FUNCTION_BLOCK _LINT_TestSuite EXTENDS TcUnit.FB_TestSuite
VAR
END_VAR

TestAddress();
TestClearReference();
TestClone();
TestTypeNameReturnsExpected();
TestIsFloat();
TestIsSigned();
TestMakeReferenceToFollowsReference();
TestMakeReferenceToUpdatesReference();
TestSize();
TestValueReturnsExpectedAfterInit();
TestValueReturnsExpectedAfterChange();
TestSerializeTypeWith();
TestSerializeWith();
TestTryDeserializeFrom();
TestTryMakeReferenceToFollowsReference();
TestTryMakeReferenceToUpdatesReference();

METHOD PUBLIC TestAddress
VAR
    _type : _LINT(0);
    notExpected : PVOID := 0;
    actual : PVOID;
END_VAR
TEST('TestAddress');

actual := _type.Address;

AssertFalse(
    Condition := (notExpected = actual),
    Message := 'Type did not return a valid address.'
);

TEST_FINISHED();
END_METHOD

METHOD PUBLIC TestClearReference
VAR
    _type : _LINT(0);
	target : LINT := 0;
    expected : LINT := 0;
    actual : LINT;
END_VAR
TEST('TestClearReference');

_type.MakeReferenceTo(target);
_type.ClearReference();
target := 123;

actual := _type.Value;

AssertEquals(
    Expected := expected,
    Actual := actual,
    Message := 'Value incorrectly followed target change'
);

TEST_FINISHED();
END_METHOD

METHOD PUBLIC TestClone
VAR
    _type : _LINT(123);
	clone : I_Datatype;
	isValidClone : BOOL;
	compareResult : DINT;
END_VAR
TEST('TestClone');

clone := _type.Clone();

isValidClone := clone <> 0;

IF isValidClone THEN
	compareResult := memcmp(_type.Address, clone.Address, clone.Size);
END_IF

AssertTrue(
	Condition := isValidClone,
	Message := 'Clone did not produce a clone'
);

AssertEquals_DINT(
	Expected := 0,
    Actual := compareResult,
    Message := 'Clone did not return a valid clone.'
);

clone.Dispose();

TEST_FINISHED();
END_METHOD

METHOD PUBLIC TestIsFloat
VAR
    _type : _LINT(0);
END_VAR
TEST('TestIsFloat');

AssertFalse(
	Condition := _type.IsFloat,
    Message := 'Type did not correctly identify itself as being unsigned'
);

TEST_FINISHED();
END_METHOD

METHOD PUBLIC TestIsSigned
VAR
    _type : _LINT(0);
END_VAR
TEST('TestIsSigned');

AssertTrue(
	Condition := _type.IsSigned,
    Message := 'Type did not correctly identify itself as being signed'
);

TEST_FINISHED();
END_METHOD

METHOD PUBLIC TestMakeReferenceToFollowsReference
VAR
    _type : _LINT(0);
	target : LINT := 0;
    expected : LINT := 123;
    actual : LINT;
END_VAR
TEST('TestMakeReferenceToFollowsReference');

_type.MakeReferenceTo(target);
target := 123;

actual := _type.Value;

AssertEquals(
    Expected := expected,
    Actual := actual,
    Message := 'Value did not follow target change'
);

TEST_FINISHED();
END_METHOD

METHOD PUBLIC TestMakeReferenceToUpdatesReference
VAR
    _type : _LINT(0);
	target : LINT := 0;
    expected : LINT := 123;
    actual : LINT;
END_VAR
TEST('TestMakeReferenceToUpdatesReference');

_type.MakeReferenceTo(target);
_type.Value := 123;

actual := target;

AssertEquals(
    Expected := expected,
    Actual := actual,
    Message := 'Value did not update target'
);

TEST_FINISHED();
END_METHOD

METHOD PUBLIC TestSerializeTypeWith
VAR
    _type : _LINT(0);
    serializer : JsonSerializer;
    expected : STRING(500) := '{"typeName":"LINT","minValue":-9223372036854775808,"maxValue":9223372036854775807,"isSigned":true,"isFloat":false}';
    actual : STRING(500);
END_VAR
TEST('TestSerializeTypeWith');

serializer.Reset();
_type.SerializeTypeWith(serializer);
serializer.TryGetSerializedData(ADR(actual), SIZEOF(actual));

AssertEquals_STRING(
    Expected := expected,
    Actual := actual,
    Message := 'Serialization of type did not return correct string.'
);

TEST_FINISHED();
END_METHOD

METHOD PUBLIC TestSerializeWith
VAR
    _type : _LINT(32767);
    serializer : JsonSerializer;
    expected : STRING := '32767';
    actual : STRING(500);
END_VAR
TEST('TestSerializeWith');

serializer.Reset();
_type.SerializeWith(serializer);
serializer.TryGetSerializedData(ADR(actual), SIZEOF(actual));

AssertEquals_STRING(
    Expected := expected,
    Actual := actual,
    Message := 'Serialization of type data did not return correct string.'
);

TEST_FINISHED();
END_METHOD

METHOD PUBLIC TestSize
VAR
    _type : _LINT(0);
    expected : UDINT := SIZEOF(LINT);
    actual : UDINT;
END_VAR
TEST('TestSize');

actual := _type.Size;

AssertEquals_UDINT(
    Expected := Expected,
    Actual := actual,
    Message := 'Type did not return the correct size.'
);

TEST_FINISHED();
END_METHOD

METHOD PUBLIC TestTryDeserializeFrom
VAR
    deserializer : JsonDeserializer;
    feedback : DeserializerFeedback;
    json : STRING := '32767';
    _type : _LINT(0);
    expected : LINT := 32767;
    actual : LINT;
 END_VAR
TEST('TestTryDeserializeFrom');

deserializer.Reset();
deserializer.TryLoad(json);
_type.TryDeserializeFrom(Deserializer, Feedback);

actual := _type.Value;

AssertEquals(
    Expected := expected,
    Actual := actual,
    Message := 'Type did not deserialize correctly.'
);

TEST_FINISHED();
END_METHOD

METHOD PUBLIC TestTryMakeReferenceToFollowsReference
VAR
    _type : _LINT(0);
	target : _LINT(0);
    expected : LINT := 123;
    actual : LINT;
END_VAR
TEST('TestTryMakeReferenceToFollowsReference');

_type.TryMakeReferenceTo(target);
target.Value := 123;

actual := _type.Value;

AssertEquals(
    Expected := expected,
    Actual := actual,
    Message := 'Value did not follow target change'
);

TEST_FINISHED();
END_METHOD

METHOD PUBLIC TestTryMakeReferenceToUpdatesReference
VAR
    _type : _LINT(0);
	target : _LINT(0);
    expected : LINT := 123;
    actual : LINT;
END_VAR
TEST('TestTryMakeReferenceToUpdatesReference');

_type.TryMakeReferenceTo(target);
_type.Value := 123;

actual := target.Value;

AssertEquals(
    Expected := expected,
    Actual := actual,
    Message := 'Value did not update target'
);

TEST_FINISHED();
END_METHOD

METHOD PUBLIC TestTypeNameReturnsExpected
VAR
    _type : _LINT(0);
    expected : STRING := 'LINT';
    actual : STRING;
END_VAR
TEST('TestTypeNameReturnsExpected');

actual := _type.TypeName;

AssertEquals_STRING(
    Expected := expected,
    Actual := actual,
    Message := 'Type did not return correct iec type.'
);

TEST_FINISHED();
END_METHOD

METHOD PUBLIC TestValueReturnsExpectedAfterChange
VAR
    _type : _LINT(0);
    expected : LINT := 32767;
    actual : LINT;
END_VAR
TEST('TestValueReturnsExpectedAfterChange');

_type.Value := 32767;

actual := _type.Value;

AssertEquals(
    Expected := expected,
    Actual := actual,
    Message := 'Expected value not returned after change.'
);

TEST_FINISHED();
END_METHOD

METHOD PUBLIC TestValueReturnsExpectedAfterInit
VAR
    _type : _LINT(32767);
    expected : LINT := 32767;
    actual : LINT;
END_VAR
TEST('TestValueReturnsExpectedAfterInit');

actual := _type.Value;

AssertEquals(
    Expected := expected,
    Actual := actual,
    Message := 'Expected value not returned after Init.'
);

TEST_FINISHED();
END_METHOD

END_FUNCTION_BLOCK

(* stored: Version 1.1.0.1, ProductVersion 3.1.4024.12
   POU _LINT_TestSuite: Id {ffc2cacf-7838-04b8-0188-c8cbaeceb051}, SpecialFunc None
   Method TestAddress: Id {96fa209b-1c3b-01f0-2361-83892fadca1e}
   Method TestClearReference: Id {bcb31aad-f7a6-058f-0132-4889f60e3a28}
   Method TestClone: Id {55139858-7e7a-043c-00ed-fa9449ef207d}
   Method TestIsFloat: Id {19633a59-7ecc-43d8-b9fd-07e68c719fe2}
   Method TestIsSigned: Id {b08a6895-bafd-0617-1282-da05443ac502}
   Method TestMakeReferenceToFollowsReference: Id {9db3bd62-8026-0717-1b49-3e66ad6dc48b}
   Method TestMakeReferenceToUpdatesReference: Id {06c34ca2-615c-0353-22e6-fde8c4860c4c}
   Method TestSerializeTypeWith: Id {d80e8f2c-736c-0c27-1419-c92f8cefd780}
   Method TestSerializeWith: Id {0434dea0-6b9d-0dfb-0cf3-214aca8bb7cc}
   Method TestSize: Id {45eea9d8-f4cd-07df-31ca-c50a808407b4}
   Method TestTryDeserializeFrom: Id {68d18972-e9c3-0d81-0fbb-bdd875d150e5}
   Method TestTryMakeReferenceToFollowsReference: Id {0dbee80a-4278-0237-1e1b-c0d52eaeb474}
   Method TestTryMakeReferenceToUpdatesReference: Id {19cab586-83c4-000c-1d47-fe00e83bf118}
   Method TestTypeNameReturnsExpected: Id {af893787-51f2-0375-1e3f-557174598dc9}
   Method TestValueReturnsExpectedAfterChange: Id {a95ad73d-32b5-046b-11d3-7715f5e5df97}
   Method TestValueReturnsExpectedAfterInit: Id {7fe5569f-9614-06ba-1442-9ca129453fe4} *)
